ABB RobotStudio station: Practica2.rsstn

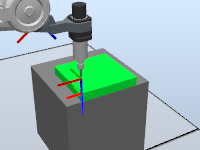
Station Practica2 (saved by RobotStudio 20.4.9280.0)
Controller Controlador3
  mechanical unit ROB_1: IRB140_6_81_C_03, 6 joints, base frame (0, 0, 0) mm
Layout (positions relative to the parent item):
  - IRB140_6_81_C_03 [mechanism, from Robots\IRB140_6_81_C_G_03.rslib] at (0, 0, 0) mm; joint values [0, -0.3449, 0.5009, 0, 0.7516, 0] (rad or m)
  - MyTool [mechanism, from Training Objects\myTool.rslib] at (363.67, 0, 580.53) mm, rotated rx 180 ry 38 rz 180 deg
  - Pieza_1 [part]
  - Pieza_8 [part]
Attachment: MyTool is attached to IRB140_6_81_C_03 / Link6
Targets, tools, work objects and paths stored in the station, written as RAPID:
! task T_ROB1
MODULE CalibData
  PERS tooldata MyTool:=[TRUE,[[31.792631019,0,229.638935148],[0.945518576,0,0.325568154,0]],[1,[0,0,1],[1,0,0,0],0,0,0]];
ENDMODULE

! task T_ROB1
MODULE Module1
  CONST robtarget Target_10:=[[480,0,330],[0,0,1,0],[0,0,0,0],[9E+09,9E+09,9E+09,9E+09,9E+09,9E+09]];
  PROC Path_10()
    MoveL Target_10,v200,z100,MyTool\WObj:=wobj0;
  ENDPROC
ENDMODULE

